TYPE ST_CalibrationReportLine :
STRUCT
	sDateTime           : STRING(40);
    sPumpNo             : STRING(10);
    sStep               : STRING(20);
    sTareWt             : STRING(30);
    sGrossWt            : STRING(30);
    sNetWt              : STRING(30);
    sNetVolume          : STRING(30);
    sTargetVolume       : STRING(30);
    sDifferencePercent  : STRING(30);
    sCriteria           : STRING(20);
    sPumpRevs           : STRING(30);
END_STRUCT
END_TYPE

(* stored: Version 1.1.0.1, ProductVersion 3.1.4024.15
   DUT ST_CalibrationReportLine: Id {e7009d4a-b484-4483-9651-008b9a344a64} *)
